TYPE T_Ctrl_SIf_MOD_Par :
STRUCT
	///[ms] wait time in pick position
	udiWaitPick_ms: UDINT;
END_STRUCT
END_TYPE

(* stored: Version 1.1.0.1, ProductVersion 3.1.0.25
   DUT T_Ctrl_SIf_MOD_Par: Id {e981b296-b9b9-4945-b7e9-494e412aed9e} *)
